INTERFACE ITF_RequestChanges EXTENDS ITF_BaseComponent

METHOD Testing : BOOL
VAR_INPUT
END_VAR
END_METHOD

END_INTERFACE

(* stored: Version 1.1.0.1
   Itf ITF_RequestChanges: Id {f1f18d3a-38da-0698-1651-a23ce385ae08}
   Method Testing: Id {76774f7f-0a54-00a4-06ca-51b2be049abf} *)
